// TIA Portal V17 export
// export: Created 2023-02-14T02:49:48.167377Z, ExportSetting WithDefaults, DisplayName Totally Integrated Automation Portal, DisplayVersion V17, DisplayName TIA Portal Openness, DisplayVersion V17, DisplayName TIA Portal Teamcenter Gateway, DisplayVersion V17, DisplayName TIA Portal Version Control Interface, DisplayVersion V17, DisplayName SINAMICS Startdrive Advanced, DisplayVersion V17, DisplayName SINAMICS Startdrive G130, G150, S120, S150, SINAMICS MV, S210, DisplayVersion V17, DisplayName SINAMICS Startdrive G110M, G120, G120C, G120D, G120P, G115D, DisplayVersion V17, DisplayName STEP 7 Professional, DisplayVersion V17, DisplayName STEP 7 Safety, DisplayVersion V17, DisplayName WinCC Professional, DisplayVersion V17
FUNCTION_BLOCK "Storage Tank"   // FB7, LAD
{ S7_Optimized_Access := 'TRUE' }
VERSION : 0.1
// stored: AutoNumber true, IsIECCheckEnabled false, IsRetainMemResEnabled false, MemoryReserve 100, SetENOAutomatically false, UDAEnableTagReadback false
   VAR_INPUT
      Lock : Bool;
      Reset : Bool;
   END_VAR
   VAR_OUTPUT
      AV_Inlet : Bool;
   END_VAR
   VAR_IN_OUT
      Tank_Level : Real;
   END_VAR
   VAR
      Parameter : Struct
         Level_High : Real := 100.0;
         Level_Med : Real := 50.0;
         Level_Low : Real;
      END_STRUCT;
      State : Struct
         Tank_HL : Bool;
         Tank_ML : Bool;
         Tank_LL : Bool;
      END_STRUCT;
      Actuator : Struct
         AV_Inlet : Bool;
      END_STRUCT;
      AlwaysOn : Bool;
      Stat_Ready_for_Transfer : Bool;
      Ready_for_Transfer : Bool;
   END_VAR
BEGIN

REGION Network 1: Always On
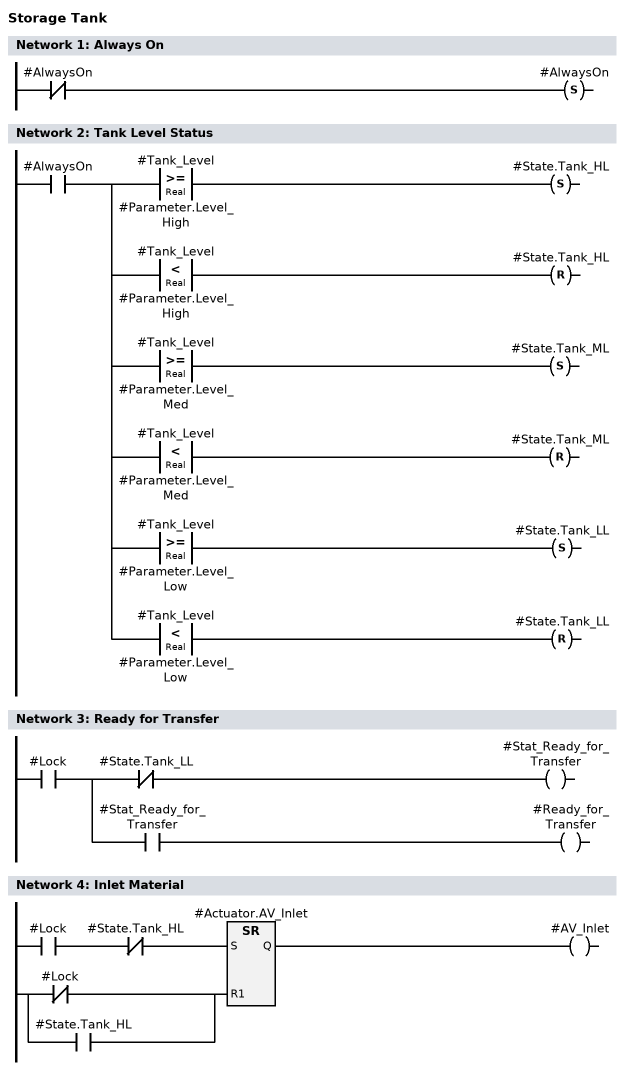
   RUNG wire#powerrail
      I_Contact( #AlwaysOn )
      S_Coil( #AlwaysOn )
   END_RUNG
   // the same network as SCL:
   IF NOT #AlwaysOn THEN #AlwaysOn := TRUE; END_IF;
END_REGION

REGION Network 2: Tank Level Status
   RUNG wire#powerrail
      Contact( #AlwaysOn )
      wire#w1
      { S7_Templates := "SrcType := Real" } GE_Contact(in1 := #Tank_Level, in2 := #Parameter.Level_High)
      S_Coil( #State.Tank_HL )
   END_RUNG
   RUNG wire#w1
      { S7_Templates := "SrcType := Real" } LT_Contact(in1 := #Tank_Level, in2 := #Parameter.Level_High)
      R_Coil( #State.Tank_HL )
   END_RUNG
   RUNG wire#w1
      { S7_Templates := "SrcType := Real" } GE_Contact(in1 := #Tank_Level, in2 := #Parameter.Level_Med)
      S_Coil( #State.Tank_ML )
   END_RUNG
   RUNG wire#w1
      { S7_Templates := "SrcType := Real" } LT_Contact(in1 := #Tank_Level, in2 := #Parameter.Level_Med)
      R_Coil( #State.Tank_ML )
   END_RUNG
   RUNG wire#w1
      { S7_Templates := "SrcType := Real" } GE_Contact(in1 := #Tank_Level, in2 := #Parameter.Level_Low)
      S_Coil( #State.Tank_LL )
   END_RUNG
   RUNG wire#w1
      { S7_Templates := "SrcType := Real" } LT_Contact(in1 := #Tank_Level, in2 := #Parameter.Level_Low)
      R_Coil( #State.Tank_LL )
   END_RUNG
   // the same network as SCL:
   IF #AlwaysOn AND (#Tank_Level >= #Parameter.Level_High) THEN #State.Tank_HL := TRUE; END_IF;
   IF #AlwaysOn AND (#Tank_Level < #Parameter.Level_High) THEN #State.Tank_HL := FALSE; END_IF;
   IF #AlwaysOn AND (#Tank_Level >= #Parameter.Level_Med) THEN #State.Tank_ML := TRUE; END_IF;
   IF #AlwaysOn AND (#Tank_Level < #Parameter.Level_Med) THEN #State.Tank_ML := FALSE; END_IF;
   IF #AlwaysOn AND (#Tank_Level >= #Parameter.Level_Low) THEN #State.Tank_LL := TRUE; END_IF;
   IF #AlwaysOn AND (#Tank_Level < #Parameter.Level_Low) THEN #State.Tank_LL := FALSE; END_IF;
END_REGION

REGION Network 3: Ready for Transfer
   RUNG wire#powerrail
      Contact( #Lock )
      wire#w1
      I_Contact( #State.Tank_LL )
      Coil( #Stat_Ready_for_Transfer )
   END_RUNG
   RUNG wire#w1
      Contact( #Stat_Ready_for_Transfer )
      Coil( #Ready_for_Transfer )
   END_RUNG
   // the same network as SCL:
   #Stat_Ready_for_Transfer := #Lock AND NOT #State.Tank_LL;
   #Ready_for_Transfer := #Lock AND #Stat_Ready_for_Transfer;
END_REGION

REGION Network 4: Inlet Material
   RUNG wire#powerrail
      Contact( #Lock )
      I_Contact( #State.Tank_HL )
      S_SR(operand := #Actuator.AV_Inlet, r1 := wire#w1)
      Coil( #AV_Inlet )
   END_RUNG
   RUNG wire#powerrail
      I_Contact( #Lock )
   END_RUNG wire#w1
   RUNG wire#powerrail
      Contact( #State.Tank_HL )
   END_RUNG wire#w1
   // the same network as SCL:
   IF #Lock AND NOT #State.Tank_HL THEN
       #Actuator.AV_Inlet := TRUE;   // SR flip-flop
   END_IF;
   IF NOT #Lock OR #State.Tank_HL THEN #Actuator.AV_Inlet := FALSE; END_IF;
   #AV_Inlet := #Actuator.AV_Inlet;
END_REGION
END_FUNCTION_BLOCK
